Staubli VAL3: CALL.pjx

--- CALL.pjx ---
Parameters version=s7.5 stackSize=5000 millimeterUnit=true
Program file=find.pgx
Program file=get.pgx
Program file=getSize.pgx
Program file=getType.pgx
Program file=load.pgx
Program file=loadIt.pgx
Program file=onEdit.pgx
Program file=onInsert.pgx
Program file=onProgEnd.pgx
Program file=onRun.pgx
Program file=onStart.pgx
Program file=onStop.pgx
Data file=CALL.dtx
Library alias=use path=Disk://kernel/userPage/userPage.pjx
Library alias=saveData path=Disk://saveData/saveData.pjx
Library alias=language path=Disk://kernel/language/language.pjx
Library alias=cycleStatus path=Disk://cycleStatus/cycleStatus.pjx
Library alias=extCall0 path=Disk://..//templates/call/call.pjx
Library alias=extCall1 path=Disk://..//templates/call/call.pjx
Library alias=extCall2 path=Disk://..//templates/call/call.pjx
Library alias=extCall3 path=Disk://..//templates/call/call.pjx
Library alias=extCall4 path=Disk://..//templates/call/call.pjx
Library alias=extCall5 path=Disk://..//templates/call/call.pjx
Library alias=extCall6 path=Disk://..//templates/call/call.pjx
Library alias=extCall7 path=Disk://..//templates/call/call.pjx
Library alias=extCall8 path=Disk://..//templates/call/call.pjx
Library alias=extCall9 path=Disk://..//templates/call/call.pjx
Library alias=extCall10 path=Disk://..//templates/call/call.pjx
Library alias=extCall11 path=Disk://..//templates/call/call.pjx
Library alias=extCall12 path=Disk://..//templates/call/call.pjx
Library alias=extCall13 path=Disk://..//templates/call/call.pjx
Library alias=extCall14 path=Disk://..//templates/call/call.pjx
Library alias=extCall15 path=Disk://..//templates/call/call.pjx
Library alias=extCall16 path=Disk://..//templates/call/call.pjx
Library alias=extCall17 path=Disk://..//templates/call/call.pjx
Library alias=extCall18 path=Disk://..//templates/call/call.pjx
Library alias=extCall19 path=Disk://..//templates/call/call.pjx

--- CALL.dtx ---
num nLoad[20]
string listCall = "_placePrinter"
public string sItems
string sCallTemp = "Disk://..//templates/call"
bool bInit
bool bMutex

--- get.pgx ---
public program get(string& x_sItem[], num x_nIndex)
begin
  x_sItem=right(listCall[x_nIndex],len(listCall[x_nIndex])-1)
end

--- getSize.pgx ---
public program getSize(num& x_nSize[])
  local num i
  local num j
begin
  //
  // search if there are Call in the Disk
  //
  libList("",listCall)
  for i=0 to (size(listCall)-1)
    if left(listCall[i],1)!="_"
      if i==size(listCall[i])-1 and i==0
        listCall=""
      else
        delete(listCall[i])
        i=i-1
      endIf
    endIf
  endFor
  if listCall!=""
    x_nSize=size(listCall)
  else
    x_nSize=0
  endIf
end

--- getType.pgx ---
program getType(string& x_sType[])
  local num l_nPos
  local string l_sPath
begin
  // get the TypePath
  l_sPath=libPath()
  do
    l_nPos=find(l_sPath,"/")
    if l_nPos==-1
      l_nPos=find(l_sPath,"\")
    endIf
    if l_nPos!=-1
      l_sPath=right(l_sPath,len(l_sPath)-l_nPos-1)
    endIf
  until l_nPos==-1
  x_sType=l_sPath
end

--- loadIt.pgx ---
program loadIt(string x_sName)
  local string l_sPath
  local num l_nTime
  local num l_nResult
  local num l_nMin
  local bool l_bLoaded
  local bool l_bOverride
  local num l_nId
  local num i
begin
  //
  l_nTime=clock()
  // MUTEX IT
  if !watch(bMutex==false,1)
    bMutex=false
    if saveData:bDebug
      logMsg("[DEBUG] MEMORY: CALL:bMutex -> TRUE FAULT")
    endIf
  endIf
  //
  setMutex(bMutex)
  // load in the memory the selected extCall
  l_sPath="Disk://"
  // MEMORY STRATEGY
  // use 19 extCall to store the extCall load
  do
    switch l_nId
      case 0
        if extCall0:libPath()==sCallTemp or extCall0:libPath()=="" or l_bOverride or (l_sPath+x_sName)==extCall0:libPath()
          if (l_sPath+x_sName)!=extCall0:libPath()
            l_nResult=extCall0:libLoad(l_sPath+x_sName)
          endIf
          if l_nResult==0
            call extCall0:start()
          endIf
          l_bLoaded=true
        endIf
      break
      case 1
        if extCall1:libPath()==sCallTemp or extCall1:libPath()=="" or l_bOverride or (l_sPath+x_sName)==extCall1:libPath()
          if (l_sPath+x_sName)!=extCall1:libPath()
            l_nResult=extCall1:libLoad(l_sPath+x_sName)
          endIf
          if l_nResult==0
            call extCall1:start()
          endIf
          l_bLoaded=true
        endIf
      break
      case 2
        if extCall2:libPath()==sCallTemp or extCall2:libPath()=="" or l_bOverride or (l_sPath+x_sName)==extCall2:libPath()
          if (l_sPath+x_sName)!=extCall2:libPath()
            l_nResult=extCall2:libLoad(l_sPath+x_sName)
          endIf
          if l_nResult==0
            call extCall2:start()
          endIf
          l_bLoaded=true
        endIf
      break
      case 3
        if extCall3:libPath()==sCallTemp or extCall3:libPath()=="" or l_bOverride or (l_sPath+x_sName)==extCall3:libPath()
          if (l_sPath+x_sName)!=extCall3:libPath()
            l_nResult=extCall3:libLoad(l_sPath+x_sName)
          endIf
          if l_nResult==0
            call extCall3:start()
          endIf
          l_bLoaded=true
        endIf
      break
      case 4
        if extCall4:libPath()==sCallTemp or extCall4:libPath()=="" or l_bOverride or (l_sPath+x_sName)==extCall4:libPath()
          if (l_sPath+x_sName)!=extCall4:libPath()
            l_nResult=extCall4:libLoad(l_sPath+x_sName)
          endIf
          if l_nResult==0
            call extCall4:start()
          endIf
          l_bLoaded=true
        endIf
      break
      case 5
        if extCall5:libPath()==sCallTemp or extCall5:libPath()=="" or l_bOverride or (l_sPath+x_sName)==extCall5:libPath()
          if (l_sPath+x_sName)!=extCall5:libPath()
            l_nResult=extCall5:libLoad(l_sPath+x_sName)
          endIf
          if l_nResult==0
            call extCall5:start()
          endIf

          l_bLoaded=true
        endIf
      break
      case 6
        if extCall6:libPath()==sCallTemp or extCall6:libPath()=="" or l_bOverride or (l_sPath+x_sName)==extCall6:libPath()
          if (l_sPath+x_sName)!=extCall6:libPath()
            l_nResult=extCall6:libLoad(l_sPath+x_sName)
          endIf
          if l_nResult==0
            call extCall6:start()
          endIf

          l_bLoaded=true
        endIf
      break
      case 7
        if extCall7:libPath()==sCallTemp or extCall7:libPath()=="" or l_bOverride or (l_sPath+x_sName)==extCall7:libPath()
          if (l_sPath+x_sName)!=extCall7:libPath()
            l_nResult=extCall7:libLoad(l_sPath+x_sName)
          endIf
          if l_nResult==0
            call extCall7:start()
          endIf
          l_bLoaded=true
        endIf
      break
      case 8
        if extCall8:libPath()==sCallTemp or extCall8:libPath()=="" or l_bOverride or (l_sPath+x_sName)==extCall8:libPath()
          if (l_sPath+x_sName)!=extCall8:libPath()
            l_nResult=extCall8:libLoad(l_sPath+x_sName)
          endIf
          if l_nResult==0
            call extCall8:start()
          endIf
          l_bLoaded=true
        endIf
      break
      case 9
        if extCall9:libPath()==sCallTemp or extCall9:libPath()=="" or l_bOverride or (l_sPath+x_sName)==extCall9:libPath()
          if (l_sPath+x_sName)!=extCall9:libPath()
            l_nResult=extCall9:libLoad(l_sPath+x_sName)
          endIf
          if l_nResult==0
            call extCall9:start()
          endIf
          l_bLoaded=true
        endIf
      break
      case 10
        if extCall10:libPath()==sCallTemp or extCall10:libPath()=="" or l_bOverride or (l_sPath+x_sName)==extCall10:libPath()
          if (l_sPath+x_sName)!=extCall10:libPath()
            l_nResult=extCall10:libLoad(l_sPath+x_sName)
          endIf
          if l_nResult==0
            call extCall10:start()
          endIf
          l_bLoaded=true
        endIf
      break
      case 11
        if extCall11:libPath()==sCallTemp or extCall11:libPath()=="" or l_bOverride or (l_sPath+x_sName)==extCall11:libPath()
          if (l_sPath+x_sName)!=extCall11:libPath()
            l_nResult=extCall11:libLoad(l_sPath+x_sName)
          endIf
          if l_nResult==0
            call extCall11:start()
          endIf
          l_bLoaded=true
        endIf
      break
      case 12
        if extCall12:libPath()==sCallTemp or extCall12:libPath()=="" or l_bOverride or (l_sPath+x_sName)==extCall12:libPath()
          if (l_sPath+x_sName)!=extCall12:libPath()
            l_nResult=extCall12:libLoad(l_sPath+x_sName)
          endIf
          if l_nResult==0
            call extCall12:start()
          endIf
          l_bLoaded=true
        endIf
      break
      case 13
        if extCall13:libPath()==sCallTemp or extCall13:libPath()=="" or l_bOverride or (l_sPath+x_sName)==extCall13:libPath()
          if (l_sPath+x_sName)!=extCall13:libPath()
            l_nResult=extCall13:libLoad(l_sPath+x_sName)
          endIf
          if l_nResult==0
            call extCall13:start()
          endIf
          l_bLoaded=true
        endIf
      break
      case 14
        if extCall14:libPath()==sCallTemp or extCall14:libPath()=="" or l_bOverride or (l_sPath+x_sName)==extCall14:libPath()
          if (l_sPath+x_sName)!=extCall14:libPath()
            l_nResult=extCall14:libLoad(l_sPath+x_sName)
          endIf
          if l_nResult==0
            call extCall14:start()
          endIf
          l_bLoaded=true
        endIf
      break
      case 15
        if extCall15:libPath()==sCallTemp or extCall15:libPath()=="" or l_bOverride or (l_sPath+x_sName)==extCall15:libPath()
          if (l_sPath+x_sName)!=extCall15:libPath()
            l_nResult=extCall15:libLoad(l_sPath+x_sName)
          endIf
          if l_nResult==0
            call extCall15:start()
          endIf
          l_bLoaded=true
        endIf
      break
      case 16
        if extCall16:libPath()==sCallTemp or extCall16:libPath()=="" or l_bOverride or (l_sPath+x_sName)==extCall16:libPath()
          if (l_sPath+x_sName)!=extCall16:libPath()
            l_nResult=extCall16:libLoad(l_sPath+x_sName)
          endIf
          if l_nResult==0
            call extCall16:start()
          endIf
          l_bLoaded=true
        endIf
      break
      case 17
        if extCall17:libPath()==sCallTemp or extCall17:libPath()=="" or l_bOverride or (l_sPath+x_sName)==extCall17:libPath()
          if (l_sPath+x_sName)!=extCall17:libPath()
            l_nResult=extCall17:libLoad(l_sPath+x_sName)
          endIf
          if l_nResult==0
            call extCall17:start()
          endIf
          l_bLoaded=true
        endIf
      break
      case 18
        if extCall18:libPath()==sCallTemp or extCall18:libPath()=="" or l_bOverride or (l_sPath+x_sName)==extCall18:libPath()
          if (l_sPath+x_sName)!=extCall18:libPath()
            l_nResult=extCall18:libLoad(l_sPath+x_sName)
          endIf
          if l_nResult==0
            call extCall18:start()
          endIf
          l_bLoaded=true
        endIf
      break
      case 19
        if extCall19:libPath()==sCallTemp or extCall19:libPath()=="" or l_bOverride or (l_sPath+x_sName)==extCall19:libPath()
          if (l_sPath+x_sName)!=extCall19:libPath()
            l_nResult=extCall19:libLoad(l_sPath+x_sName)
          endIf
          if l_nResult==0
            call extCall19:start()
          endIf
          l_bLoaded=true
        endIf
      break
    endSwitch
    //
    if !l_bLoaded
      if l_nId>=19
        // check for the less use
        l_nMin=nLoad
        l_bOverride=true
        for i=0 to 19
          if nLoad[l_nId]<=l_nMin
            l_nId=i
          endIf
        endFor
      else
        //increase
        l_nId=l_nId+1
      endIf
    endIf
    //
    // exit
    //
    delay(0)
  until l_bLoaded
  //
  // validate
  //
  if l_bOverride
    nLoad[l_nId]=1
  else
    nLoad[l_nId]=nLoad[l_nId]+1
  endIf
  if l_nResult!=0
    logMsg("[DEBUG] MEMORY:Charged "+x_sName+" error code: "+toString("",l_nResult))
  endIf
  // release
  bMutex=false
end

--- onEdit.pgx ---
public program onEdit(string& x_sItem[])
  local string l_sEvent
  local num l_nSize
  local num i
  local num l_nKey
  local string l_sType
begin
  cls()
  call language:message(l_sEvent,64)
  call use:clear(0,13)
  call use:typeCenter(13,l_sEvent,40,true)
  x_sItem=""
  call use:setSizeList(19,0,19,11)
  call getType(l_sType)
  call use:listcreate(l_sType+" ")
  call getSize(l_nSize)
  if l_nSize!=0
    for i=0 to l_nSize-1
      call get(l_sEvent,i)
      call use:listadd(l_sEvent)
    endFor
    call use:listupdate(0)
    do
      l_nKey=get()
      call use:listevent(l_nKey,i,l_sEvent)
    until l_nKey==255 or l_nKey==270
    if l_nKey==270
      x_sItem=l_sEvent
    endIf
  endIf
  call use:nullKey(l_nKey)
end

--- onInsert.pgx ---
public program onInsert(string& x_sItem[])
  local num l_nSize
  local num i
  local string l_sEvent
  local num l_nKey
  local string l_sType
begin
  cls()
  call language:message(l_sEvent,64)
  call use:clear(0,13)
  call use:typeCenter(13,l_sEvent,40,true)
  x_sItem=""
  call use:setSizeList(19,0,19,11)
  call getType(l_sType)
  call use:listcreate(l_sType+" ")
  call getSize(l_nSize)
  if l_nSize!=0
    for i=0 to l_nSize-1
      call get(l_sEvent,i)
      call use:listadd(l_sEvent)
    endFor
    call use:listupdate(0)
    do
      l_nKey=get()
      call use:listevent(l_nKey,i,l_sEvent)
    until l_nKey==255 or l_nKey==270
    if l_nKey==270
      x_sItem=l_sEvent
    endIf
  endIf
  call use:nullKey(l_nKey)
end

--- onRun.pgx ---
public program onRun(string& x_sItem[])
  local num l_nResult
begin
  //
  call loadIt("_"+x_sItem)
  //
end

--- onStart.pgx ---
public program onStart(string& x_sItem[])
begin
  // init all
  bInit=true
end

--- onStop.pgx ---
public program onStop(string& x_sItem[])
  local num l_nResult
begin
  // reload all the template
  l_nResult=extCall0:libLoad("Disk://..//templates/call")
  delay(0)
  l_nResult=l_nResult+extCall1:libLoad("Disk://..//templates/call")
  delay(0)
  l_nResult=l_nResult+extCall2:libLoad("Disk://..//templates/call")
  delay(0)
  l_nResult=l_nResult+extCall3:libLoad("Disk://..//templates/call")
  delay(0)
  l_nResult=l_nResult+extCall4:libLoad("Disk://..//templates/call")
  delay(0)
  l_nResult=l_nResult+extCall5:libLoad("Disk://..//templates/call")
  delay(0)
  l_nResult=l_nResult+extCall6:libLoad("Disk://..//templates/call")
  delay(0)
  l_nResult=l_nResult+extCall7:libLoad("Disk://..//templates/call")
  delay(0)
  l_nResult=l_nResult+extCall8:libLoad("Disk://..//templates/call")
  delay(0)
  l_nResult=l_nResult+extCall9:libLoad("Disk://..//templates/call")
  delay(0)
  l_nResult=l_nResult+extCall10:libLoad("Disk://..//templates/call")
  delay(0)
  l_nResult=l_nResult+extCall11:libLoad("Disk://..//templates/call")
  delay(0)
  l_nResult=l_nResult+extCall12:libLoad("Disk://..//templates/call")
  delay(0)
  l_nResult=l_nResult+extCall13:libLoad("Disk://..//templates/call")
  delay(0)
  l_nResult=l_nResult+extCall14:libLoad("Disk://..//templates/call")
  delay(0)
  l_nResult=l_nResult+extCall15:libLoad("Disk://..//templates/call")
  delay(0)
  l_nResult=l_nResult+extCall16:libLoad("Disk://..//templates/call")
  delay(0)
  l_nResult=l_nResult+extCall17:libLoad("Disk://..//templates/call")
  delay(0)
  l_nResult=l_nResult+extCall18:libLoad("Disk://..//templates/call")
  delay(0)
  l_nResult=l_nResult+extCall19:libLoad("Disk://..//templates/call")
  delay(0)
end
